FUNCTION_BLOCK TcoContextBuilder IMPLEMENTS ITcoContexBuilder

METHOD Build : ITcoContexBuilder
VAR_INPUT
END_VAR
END_METHOD

METHOD FB_init : BOOL
VAR_INPUT
	bInitRetains : BOOL; // if TRUE, the retain variables are initialized (warm start / cold start)
	bInCopyCode : BOOL;  // if TRUE, the instance afterwards gets moved into the copy code (online change)	
	Context : ITcoContext; 
END_VAR
END_METHOD

METHOD WithLogger : ITcoContexBuilder
VAR_INPUT
END_VAR
END_METHOD

END_FUNCTION_BLOCK

(* stored: Version 1.1.0.1, ProductVersion 3.1.4024.9
   POU TcoContextBuilder: Id {11fcb5e1-103e-0f9c-0257-e5ca5502dbf8}, SpecialFunc None
   Method Build: Id {7331aaf2-9e6a-0ef8-0818-7d0782751f80}
   Method FB_init: Id {e931dbe5-856c-06ff-272d-79b39b5e89f4}
   Method WithLogger: Id {1658510a-bf2a-04c6-0ec2-27e989db34d1} *)
